Universal Robots PolyScope program: weigh_single_new1.urp

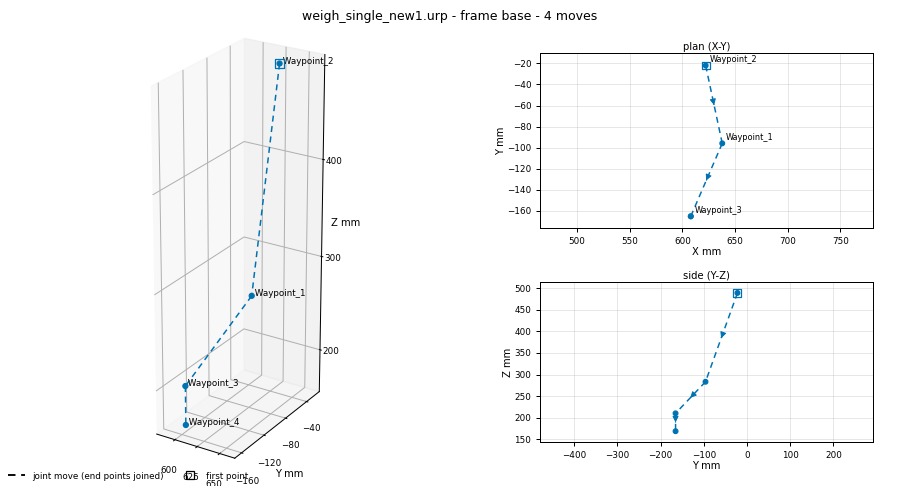
[picture p0: tool path of weigh_single_new1.urp in frame base, 4 of 4 moves have a stored position in this frame; points joined in program order, loops and branches not executed]
Program weigh_single_new1 (installation=default directory=/programs/Nicolas_Arteaga/quality createdIn=5.12.4.1101661 lastSavedIn=5.12.4.1101661 robotSerialNumber=20225502378)
Calibrated DH parameters: a=[0.00022, -0.425328, -0.389701, 0.000059, 0.000065, 0]; d=[0.162608, 0.803456, 9.992211, -10.662202, 0.099702, 0.099559]; alpha=[1.570756, 0.001543, 0.004316, 1.570651, -1.570122, 0]; deltaTheta=[0, 0.002917, 0.116094, -0.119008, 0, -0.000001]
Robot Program (runOnlyOnce=true)
  MoveJ speed 60 deg/s, acceleration 80 deg/s^2 (useActiveTCP=true) feature=Base
    Waypoint Waypoint_2: TCP in base x=622.09 y=-21.999 z=488.949 mm, rx=0.729 ry=1.5781 rz=1.7949 rad; joints [135.515, -94.567, 106.176, -67.801, 9.2, 55.784] deg; TCP offset x=0 y=0 z=191.5 mm, rx=0 ry=0 rz=0 rad
    Waypoint Waypoint_1: TCP in base x=637.825 y=-95.931 z=283.355 mm, rx=1.2165 ry=1.151 rz=1.1657 rad; joints [145.529, -90.424, 122.897, -34.058, 59.252, 0.492] deg
    Waypoint Waypoint_3: TCP in base x=607.929 y=-165.259 z=210.32 mm, rx=1.2164 ry=1.151 rz=1.1657 rad; joints [132.864, -83.639, 129.414, -47.669, 46.63, 0.933] deg
    Waypoint Waypoint_4: TCP in base x=607.939 y=-165.205 z=168.973 mm, rx=1.2164 ry=1.1511 rz=1.1658 rad; joints [132.859, -78.034, 131.663, -55.503, 46.638, 0.907] deg
    URCap Gripper (Robotiq_Grippers, Robotiq Inc.) dataModel(position=41.96078431372549, force=100.0, speed=100.0, positionInDouble=41.96078431372549, forceInDouble=100.0, speedInDouble=100.0, slaveIds=[9], blocking=true)
